DATA_BLOCK "FF_IO"
{ S7_Optimized_Access := 'FALSE' }
VERSION : 0.1
NON_RETAIN
   VAR
      BeltRotate : Bool;      // belt.rotate (PLC writes) run the belt
      EmitterEmit : Bool;     // emitter.emit (PLC writes) rising edge = feed one carton; hold each level well over one poll
      GateDivert : Bool;      // gate.divert (PLC writes) swing the blade across the lane (45 deg); FALSE parks it along the edge
      PanelGreen : Bool;      // panel.green (PLC writes) green lamp on the panel
      PanelRed : Bool;        // panel.red (PLC writes) red lamp on the panel
      PanelSetpoint : Real;   // panel.setpoint (PLC reads) the operator's pot, 4..10 s (starts at 6)
      ShortCountCount : DInt; // short_count.count (PLC reads) cartons this remover has taken off the line, running total
      TallCountCount : DInt;  // tall_count.count (PLC reads) cartons this remover has taken off the line, running total
      BeltFault : Bool;       // belt.fault (PLC reads) drive fault: TRUE = faulted; a faulted drive does not turn, whatever it is told
      EntryEyeDetect : Bool;  // entry_eye.detect (PLC reads) TRUE while anything breaks the beam to the reflector
      GateDiverted : Bool;    // gate.diverted (PLC reads) blade fully across -- a carton meeting it now is turned, not hit
      GateFault : Bool;       // gate.fault (PLC reads) drive fault: TRUE = seized; the blade stays where it is, at neither limit mid-swing
      GateHome : Bool;        // gate.home (PLC reads) blade parked along the belt edge
      PanelEstop : Bool;      // panel.estop (PLC reads) E-stop, normally closed: TRUE = healthy, FALSE = pressed; stays pressed until pulled out
      PanelReset : Bool;      // panel.reset (PLC reads) Reset button, momentary: a short pulse per press
      PanelStart : Bool;      // panel.start (PLC reads) Start button, momentary: a short pulse per press -- latch it
      PanelStop : Bool;       // panel.stop (PLC reads) Stop button, momentary: a short pulse per press
      TallEyeDetect : Bool;   // tall_eye.detect (PLC reads) TRUE while anything breaks the beam to the reflector
   END_VAR


BEGIN

END_DATA_BLOCK


FUNCTION_BLOCK "PivotDivert"
{ S7_Optimized_Access := 'TRUE' }
VERSION : 0.1

// ---------------------------------------------------------------------------
// FactoryForge starter -- Pivot diverter line (scene pivot-divert)
// Generated by tools/gen_starters.py; see README.md beside this file.
//
// THE TASK
//   Run the belt and emit a carton every panel.setpoint seconds. Two beams
//   cross the belt at the same place: entry_eye, low, sees every carton,
//   and tall_eye, high, sees only the tall ones. Every tall carton goes
//   into the chute and every short one runs on to the end. Swing the blade
//   across (gate.divert) as soon as tall_eye sees a tall carton, and hold
//   it there until tall_count.count says the carton has arrived in the
//   chute -- then home it for the short one behind. A turned carton slides
//   along the blade, driven only by the belt under it: it is off the belt
//   after about two metres of belt travel past the eyes, which at a slower
//   belt takes longer.
//
// DONE WHEN
//   Tall cartons slide along the blade into the chute and short ones pass
//   the parked blade, with the belt running the whole time. Slow the belt
//   (its Belt Speed slider) and nothing changes but the spacing: a blade
//   homed on a timer set at the rated speed lets a tall carton go half way
//   along it, and it rides on to the end. Drive gate.divert straight from
//   tall_eye.detect and the blade is home again before the carton gets
//   there. Swing the blade out only when the carton reaches it, as you
//   would fire a pusher, and it still lands in the chute -- because the
//   blade hit it. Seize the drive (gate.fault) mid-swing and neither
//   gate.home nor gate.diverted is made.
//
// Every signal is a member of the global DB "FF_IO" above: read and write
// them as "FF_IO".<Name>, e.g. "FF_IO".BeltRotate. Its comments say which
// way each one runs. Call this block from OB1 (drag it into Main; TIA creates
// the instance DB).
// ---------------------------------------------------------------------------

BEGIN

    // Your program.

END_FUNCTION_BLOCK
